TYPE ST_ITC_ElementCommands :
(**************************************************************************************
 * 	Application		:	BoxControl Framework
 *	Revision		:	$Revision: 404529 $
 *	Revision date	:	$Date: 2018-04-23 08:21:38 +0200 (Mo., 23 Apr 2018) $
 *	Last changed by	:	$Author: b7bolm $
 *	URL				:	$URL: http://almscdc.swisslog.com/repo/SWPD/Development/BoxControlFramework/20_Release/trunk/01_Software/BCF/BCF/JumpStart/20_Product/10_App/13_Elements/10_Lib/10_Conv/01_DUTs/ST_ITC_ElementCommands.TcDUT $
 *
 *	Purpose			:	Internal ITC element commands
 *
 * ------------------------------------------------------------------------------------
 *	Copyright Swisslog [IP AG], Switzerland. All rights reserved.
 * 
 * ------------------------------------------------------------------------------------
 *	
 * 	Revision History: 
 *
 * 	VERSION			DATE			INITIALS			DESCRIPTION
 *	0.1				01.01.2001		swl					Example
 *
 **************************************************************************************)
STRUCT
	StatusReport		: BOOL; // Command to send StatusReport 
	ControlReport		: BOOL; // Command to send ControlReport 
	NoErrorReport		: BOOL; // Command to send a 'no error' report
	ManualControlReport	: BOOL; // Command to send a manual control report
END_STRUCT
END_TYPE

(* stored: Version 1.1.0.1, ProductVersion 3.1.4022.12
   DUT ST_ITC_ElementCommands: Id {5c1b620c-7be2-46b6-982e-e5483d4993b9} *)
